(* IEC 61131-3 sources: SRCI/RobotLibrary/Library/Functions/Convert, 17 files *)

(* ---- ByteToFragmentAction.st ---- *)
FUNCTION ByteToFragmentAction : FragmentAction
// -------------------------------------------------------------------------
//  SRCI Robot Library
// -------------------------------------------------------------------------
//
//  Object:      FragmentActionToByte
//  Author:      Thorsten Brach
//  Date:        2024-11-05
//
//  Description:
//
//
//  Copyright:
//    (C) 2024 Thorsten Brach. All rights reserved
//             Licensed under the LGPL-3.0 license.
//
//  Disclaimer:
//    This project is provided without any guarantee and can be used for
//    private and commercial purposes. Any use is at the user’s
//    own risk and responsibility.
//
// -------------------------------------------------------------------------
VAR_INPUT
  FragmentAction : BYTE;
END_VAR

  ByteToFragmentAction.Complete:= FragmentAction.0;
  ByteToFragmentAction.Reset   := FragmentAction.1;
  ByteToFragmentAction.Clear   := FragmentAction.2;
  ByteToFragmentAction.BIT03   := FragmentAction.3;
  ByteToFragmentAction.BIT04   := FragmentAction.4;
  ByteToFragmentAction.BIT05   := FragmentAction.5;
  ByteToFragmentAction.BIT06   := FragmentAction.6;
  ByteToFragmentAction.BIT07   := FragmentAction.7;

END_FUNCTION

(* ---- CmdMessageStateToString.st ---- *)
FUNCTION CmdMessageStateToString : STRING
// -------------------------------------------------------------------------
//  SRCI Robot Library
// -------------------------------------------------------------------------
//
//  Object:      CmdMessageStateToString
//  Author:      Thorsten Brach
//  Date:        2024-11-16
//
//  Description:
//
//
//  Copyright:
//    (C) 2024 Thorsten Brach. All rights reserved
//             Licensed under the LGPL-3.0 license.
//
//  Disclaimer:
//    This project is provided without any guarantee and can be used for
//    private and commercial purposes. Any use is at the user’s
//    own risk and responsibility.
//
// -------------------------------------------------------------------------
VAR_INPUT
  /// Command message state
  Value : CmdMessageState;
END_VAR

  CASE Value
  OF
    CmdMessageState.EMPTY               : CmdMessageStateToString := StrReplace('EMPTY ({0})'              ,'{0}', USINT_TO_STRING(CmdMessageState.EMPTY));
    CmdMessageState.CREATED             : CmdMessageStateToString := StrReplace('CREATED ({0})'            ,'{0}', USINT_TO_STRING(CmdMessageState.CREATED));
    CmdMessageState.BUFFERED            : CmdMessageStateToString := StrReplace('BUFFERED ({0})'           ,'{0}', USINT_TO_STRING(CmdMessageState.BUFFERED));
    CmdMessageState.BUFFERED_IN_PLANNER : CmdMessageStateToString := StrReplace('BUFFERED_IN_PLANNER ({0})','{0}', USINT_TO_STRING(CmdMessageState.BUFFERED_IN_PLANNER));
    CmdMessageState.ACTIVE              : CmdMessageStateToString := StrReplace('ACTIVE ({0})'             ,'{0}', USINT_TO_STRING(CmdMessageState.ACTIVE));
    CmdMessageState.INTERRUPTED         : CmdMessageStateToString := StrReplace('INTERRUPTED ({0})'        ,'{0}', USINT_TO_STRING(CmdMessageState.INTERRUPTED));
    CmdMessageState.ABORT_REQUEST       : CmdMessageStateToString := StrReplace('ABORT_REQUEST ({0})'      ,'{0}', USINT_TO_STRING(CmdMessageState.ABORT_REQUEST));
    CmdMessageState.DONE                : CmdMessageStateToString := StrReplace('DONE ({0})'               ,'{0}', USINT_TO_STRING(CmdMessageState.DONE));
    CmdMessageState.ABORTED             : CmdMessageStateToString := StrReplace('ABORTED ({0})'            ,'{0}', USINT_TO_STRING(CmdMessageState.ABORTED));
    CmdMessageState.ERROR               : CmdMessageStateToString := StrReplace('ERROR ({0})'              ,'{0}', USINT_TO_STRING(CmdMessageState.ERROR));
  ELSE
    CmdMessageStateToString := CONCAT('CmdMessageStateToString-Function: Error -> no parsing for value ', USINT_TO_STRING(Value));
  END_CASE

END_FUNCTION

(* ---- CmdTypeToString.st ---- *)
FUNCTION CmdTypeToString : String
// -------------------------------------------------------------------------
//  SRCI Robot Library
// -------------------------------------------------------------------------
//
//  Object:      CmdTypeToString
//  Author:      Thorsten Brach
//  Date:        2024-11-16
//
//  Description:
//
//
//  Copyright:
//    (C) 2024 Thorsten Brach. All rights reserved
//             Licensed under the LGPL-3.0 license.
//
//  Disclaimer:
//    This project is provided without any guarantee and can be used for
//    private and commercial purposes. Any use is at the user’s
//    own risk and responsibility.
//
// -------------------------------------------------------------------------
VAR_INPUT
  /// command type
  Value : CmdType;
END_VAR

  CASE Value
  OF
    CmdType.RobotTask                   : CmdTypeToString := StrReplace('RobotTask ({0})','{0}'                  , UINT_TO_STRING(CmdType.RobotTask));

    CmdType.ReadRobotData               : CmdTypeToString := StrReplace('ReadRobotData ({0})','{0}'              , UINT_TO_STRING(CmdType.ReadRobotData));

    CmdType.EnableRobot                 : CmdTypeToString := StrReplace('EnableRobot ({0})','{0}'                , UINT_TO_STRING(CmdType.EnableRobot));

    CmdType.GroupReset                  : CmdTypeToString := StrReplace('GroupReset ({0})','{0}'                 , UINT_TO_STRING(CmdType.GroupReset));

    CmdType.ReadActualPosition          : CmdTypeToString := StrReplace('ReadActualPosition ({0})','{0}'         , UINT_TO_STRING(CmdType.ReadActualPosition));

    CmdType.ReadActualPositionCyclic    : CmdTypeToString := StrReplace('ReadActualPositionCyclic ({0})','{0}'   , UINT_TO_STRING(CmdType.ReadActualPositionCyclic));

    CmdType.ReadDHParameter             : CmdTypeToString := StrReplace('ReadDHParameter ({0})','{0}'            , UINT_TO_STRING(CmdType.ReadDHParameter));

    CmdType.RestartController           : CmdTypeToString := StrReplace('RestartController ({0})','{0}'          , UINT_TO_STRING(CmdType.RestartController));

    CmdType.ReadActualTCPVelocity       : CmdTypeToString := StrReplace('ReadActualTCPVelocity ({0})','{0}'      , UINT_TO_STRING(CmdType.ReadActualTCPVelocity));

    CmdType.UserLogin                   : CmdTypeToString := StrReplace('UserLogin ({0})','{0}'                  , UINT_TO_STRING(CmdType.UserLogin));

    CmdType.SwitchLanguage              : CmdTypeToString := StrReplace('SwitchLanguage ({0})','{0}'             , UINT_TO_STRING(CmdType.SwitchLanguage));

    CmdType.ExchangeConfiguration       : CmdTypeToString := StrReplace('ExchangeConfiguration ({0})','{0}'      , UINT_TO_STRING(CmdType.ExchangeConfiguration));

    CmdType.SetSequence                 : CmdTypeToString := StrReplace('SetSequence ({0})','{0}'                , UINT_TO_STRING(CmdType.SetSequence));

    CmdType.ChangeSpeedOverride         : CmdTypeToString := StrReplace('ChangeSpeedOverride ({0})','{0}'        , UINT_TO_STRING(CmdType.ChangeSpeedOverride));

    CmdType.ReadMessages                : CmdTypeToString := StrReplace('ReadMessages ({0})','{0}'               , UINT_TO_STRING(CmdType.ReadMessages));

    CmdType.ReadRobotReferenceDynamics  : CmdTypeToString := StrReplace('ReadRobotReferenceDynamics ({0})','{0}' , UINT_TO_STRING(CmdType.ReadRobotReferenceDynamics));

    CmdType.WriteFrameData              : CmdTypeToString := StrReplace('WriteFrameData ({0})','{0}'             , UINT_TO_STRING(CmdType.WriteFrameData));

    CmdType.WriteToolData               : CmdTypeToString := StrReplace('WriteToolData ({0})','{0}'              , UINT_TO_STRING(CmdType.WriteToolData));

    CmdType.WriteLoadData               : CmdTypeToString := StrReplace('WriteLoadData ({0})','{0}'              , UINT_TO_STRING(CmdType.WriteLoadData));

    CmdType.WriteRobotReferenceDynamics : CmdTypeToString := StrReplace('WriteRobotReferenceDynamics ({0})','{0}', UINT_TO_STRING(CmdType.WriteRobotReferenceDynamics));

    CmdType.WriteRobotDefaultDynamics   : CmdTypeToString := StrReplace('WriteRobotDefaultDynamics ({0})'  ,'{0}', UINT_TO_STRING(CmdType.WriteRobotDefaultDynamics));

    CmdType.ReadRobotDefaultDynamics    : CmdTypeToString := StrReplace('ReadRobotDefaultDynamics ({0})'   ,'{0}', UINT_TO_STRING(CmdType.ReadRobotDefaultDynamics));

    CmdType.ReadFrameData               : CmdTypeToString := StrReplace('ReadFrameData ({0})'              ,'{0}', UINT_TO_STRING(CmdType.ReadFrameData));

    CmdType.ReadToolData                : CmdTypeToString := StrReplace('ReadToolData ({0})','{0}'               , UINT_TO_STRING(CmdType.ReadToolData));

    CmdType.ReadLoadData                : CmdTypeToString := StrReplace('ReadLoadData ({0})','{0}'               , UINT_TO_STRING(CmdType.ReadLoadData));

    CmdType.ReadRobotSWLimits           : CmdTypeToString := StrReplace('ReadRobotSWLimits ({0})','{0}'          , UINT_TO_STRING(CmdType.ReadRobotSWLimits));

    CmdType.WriteRobotSWLimits          : CmdTypeToString := StrReplace('WriteRobotSWLimits ({0})','{0}'         , UINT_TO_STRING(CmdType.WriteRobotSWLimits));

    CmdType.SetOperationMode            : CmdTypeToString := StrReplace('SetOperationMode ({0})','{0}'           , UINT_TO_STRING(CmdType.SetOperationMode));

    CmdType.ReadWorkArea                : CmdTypeToString := StrReplace('ReadWorkArea ({0})','{0}'               , UINT_TO_STRING(CmdType.ReadWorkArea));

    CmdType.WriteWorkArea               : CmdTypeToString := StrReplace('WriteWorkArea ({0})','{0}'              , UINT_TO_STRING(CmdType.WriteWorkArea));

    CmdType.ActivateWorkArea            : CmdTypeToString := StrReplace('ActivateWorkArea ({0})','{0}'           , UINT_TO_STRING(CmdType.ActivateWorkArea));

    CmdType.MonitorWorkArea             : CmdTypeToString := StrReplace('MonitorWorkArea ({0})','{0}'            , UINT_TO_STRING(CmdType.MonitorWorkArea));

    CmdType.GroupJog                    : CmdTypeToString := StrReplace('GroupJog ({0})','{0}'                   , UINT_TO_STRING(CmdType.GroupJog));

    CmdType.MoveLinearAbsolute          : CmdTypeToString := StrReplace('MoveLinearAbsolute ({0})','{0}'         , UINT_TO_STRING(CmdType.MoveLinearAbsolute));

    CmdType.MoveDirectAbsolute          : CmdTypeToString := StrReplace('MoveDirectAbsolute ({0})','{0}'         , UINT_TO_STRING(CmdType.MoveDirectAbsolute));

    CmdType.MoveAxesAbsolute            : CmdTypeToString := StrReplace('MoveAxesAbsolute ({0})','{0}'           , UINT_TO_STRING(CmdType.MoveAxesAbsolute));

    CmdType.GroupStop                   : CmdTypeToString := StrReplace('GroupStop ({0})','{0}'                  , UINT_TO_STRING(CmdType.GroupStop));

    CmdType.GroupInterrupt              : CmdTypeToString := StrReplace('GroupInterrupt ({0})','{0}'             , UINT_TO_STRING(CmdType.GroupInterrupt));

    CmdType.GroupContinue               : CmdTypeToString := StrReplace('GroupContinue ({0})','{0}'              , UINT_TO_STRING(CmdType.GroupContinue));

    CmdType.MoveLinearRelative          : CmdTypeToString := StrReplace('MoveLinearRelative ({0})','{0}'         , UINT_TO_STRING(CmdType.MoveLinearRelative));

    CmdType.MoveDirectRelative          : CmdTypeToString := StrReplace('MoveDirectRelative ({0})','{0}'         , UINT_TO_STRING(CmdType.MoveDirectRelative));

    CmdType.MoveAxesRelative            : CmdTypeToString := StrReplace('MoveAxesRelative ({0})','{0}'           , UINT_TO_STRING(CmdType.MoveAxesRelative));

    CmdType.ReturnToPrimary             : CmdTypeToString := StrReplace('ReturnToPrimary ({0})','{0}'            , UINT_TO_STRING(CmdType.ReturnToPrimary));

    CmdType.MoveCircularAbsolute        : CmdTypeToString := StrReplace('MoveCircularAbsolute ({0})','{0}'       , UINT_TO_STRING(CmdType.MoveCircularAbsolute));

    CmdType.MoveCircularRelative        : CmdTypeToString := StrReplace('MoveCircularRelative ({0})','{0}'       , UINT_TO_STRING(CmdType.MoveCircularRelative));

    CmdType.MoveLinearOffset            : CmdTypeToString := StrReplace('MoveLinearOffset ({0})','{0}'           , UINT_TO_STRING(CmdType.MoveLinearOffset));

    CmdType.MoveDirectOffset            : CmdTypeToString := StrReplace('MoveDirectOffset ({0})','{0}'           , UINT_TO_STRING(CmdType.MoveDirectOffset));

    CmdType.WaitTime                    : CmdTypeToString := StrReplace('WaitTime ({0})','{0}'                   , UINT_TO_STRING(CmdType.WaitTime));

    CmdType.MoveApproachLinear          : CmdTypeToString := StrReplace('MoveApproachLinear ({0})','{0}'         , UINT_TO_STRING(CmdType.MoveApproachLinear));

    CmdType.MoveDepartLinear            : CmdTypeToString := StrReplace('MoveDepartLinear ({0})','{0}'           , UINT_TO_STRING(CmdType.MoveDepartLinear));

    CmdType.MoveApproachDirect          : CmdTypeToString := StrReplace('MoveApproachDirect ({0})','{0}'         , UINT_TO_STRING(CmdType.MoveApproachDirect));

    CmdType.MoveDepartDirect            : CmdTypeToString := StrReplace('MoveDepartDirect ({0})','{0}'           , UINT_TO_STRING(CmdType.MoveDepartDirect));

    CmdType.SearchHardstop              : CmdTypeToString := StrReplace('SearchHardstop ({0})','{0}'             , UINT_TO_STRING(CmdType.SearchHardstop));

    CmdType.SearchHardstopJ             : CmdTypeToString := StrReplace('SearchHardstopJ ({0})','{0}'            , UINT_TO_STRING(CmdType.SearchHardstopJ));

    CmdType.MovePickPlaceLinear         : CmdTypeToString := StrReplace('MovePickPlaceLinear ({0})','{0}'        , UINT_TO_STRING(CmdType.MovePickPlaceLinear));

    CmdType.MovePickPlaceDirect         : CmdTypeToString := StrReplace('MovePickPlaceDirect ({0})','{0}'        , UINT_TO_STRING(CmdType.MovePickPlaceDirect));

    CmdType.ActivateConveyorTracking    : CmdTypeToString := StrReplace('ActivateConveyorTracking ({0})','{0}'   , UINT_TO_STRING(CmdType.ActivateConveyorTracking));

    CmdType.RedefineTrackingPos         : CmdTypeToString := StrReplace('RedefineTrackingPos ({0})','{0}'        , UINT_TO_STRING(CmdType.RedefineTrackingPos));

    CmdType.SyncToConveyor              : CmdTypeToString := StrReplace('SyncToConveyor ({0})','{0}'             , UINT_TO_STRING(CmdType.SyncToConveyor));

    CmdType.ConfigureConveyor           : CmdTypeToString := StrReplace('ConfigureConveyor ({0})','{0}'          , UINT_TO_STRING(CmdType.ConfigureConveyor));

    CmdType.MoveSuperImposed            : CmdTypeToString := StrReplace('MoveSuperImposed ({0})','{0}'           , UINT_TO_STRING(CmdType.MoveSuperImposed));

    CmdType.MoveSuperImposedDynamic     : CmdTypeToString := StrReplace('MoveSuperImposedDynamic ({0})','{0}'    , UINT_TO_STRING(CmdType.MoveSuperImposedDynamic));

    CmdType.ReadDigitalInputs           : CmdTypeToString := StrReplace('ReadDigitalInputs ({0})','{0}'          , UINT_TO_STRING(CmdType.ReadDigitalInputs));

    CmdType.ReadDigitalOutputs          : CmdTypeToString := StrReplace('ReadDigitalOutputs ({0})','{0}'         , UINT_TO_STRING(CmdType.ReadDigitalOutputs));

    CmdType.WriteDigitalOutputs         : CmdTypeToString := StrReplace('WriteDigitalOutputs ({0})','{0}'        , UINT_TO_STRING(CmdType.WriteDigitalOutputs));

    CmdType.ReadIntegers                : CmdTypeToString := StrReplace('ReadIntegers ({0})','{0}'               , UINT_TO_STRING(CmdType.ReadIntegers));

    CmdType.ReadReals                   : CmdTypeToString := StrReplace('ReadReals ({0})','{0}'                  , UINT_TO_STRING(CmdType.ReadReals));

    CmdType.WriteIntegers               : CmdTypeToString := StrReplace('WriteIntegers ({0})','{0}'              , UINT_TO_STRING(CmdType.WriteIntegers));

    CmdType.WriteReals                  : CmdTypeToString := StrReplace('WriteReals ({0})','{0}'                 , UINT_TO_STRING(CmdType.WriteReals));

    CmdType.MoveLinearCam               : CmdTypeToString := StrReplace('MoveLinearCam ({0})','{0}'              , UINT_TO_STRING(CmdType.MoveLinearCam));

    CmdType.MoveDirectCam               : CmdTypeToString := StrReplace('MoveDirectCam ({0})','{0}'              , UINT_TO_STRING(CmdType.MoveDirectCam));

    CmdType.MoveCircularCam             : CmdTypeToString := StrReplace('MoveCircularCam ({0})','{0}'            , UINT_TO_STRING(CmdType.MoveCircularCam));

    CmdType.ReadAnalogInput             : CmdTypeToString := StrReplace('ReadAnalogInput ({0})','{0}'            , UINT_TO_STRING(CmdType.ReadAnalogInput));

    CmdType.ReadAnalogOutput            : CmdTypeToString := StrReplace('ReadAnalogOutput ({0})','{0}'           , UINT_TO_STRING(CmdType.ReadAnalogOutput));

    CmdType.WriteAnalogOutput           : CmdTypeToString := StrReplace('WriteAnalogOutput ({0})','{0}'          , UINT_TO_STRING(CmdType.WriteAnalogOutput));

    CmdType.MeasuringInput              : CmdTypeToString := StrReplace('MeasuringInput ({0})','{0}'             , UINT_TO_STRING(CmdType.MeasuringInput));

    CmdType.AbortMeasuringInput         : CmdTypeToString := StrReplace('AbortMeasuringInput ({0})','{0}'        , UINT_TO_STRING(CmdType.AbortMeasuringInput));

    CmdType.SetTriggerRegister          : CmdTypeToString := StrReplace('SetTriggerRegister ({0})','{0}'         , UINT_TO_STRING(CmdType.SetTriggerRegister));

    CmdType.SetTriggerLimit             : CmdTypeToString := StrReplace('SetTriggerLimit ({0})','{0}'            , UINT_TO_STRING(CmdType.SetTriggerLimit));

    CmdType.SetTriggerUser              : CmdTypeToString := StrReplace('SetTriggerUser ({0})','{0}'             , UINT_TO_STRING(CmdType.SetTriggerUser));

    CmdType.SetTriggerError             : CmdTypeToString := StrReplace('SetTriggerError ({0})','{0}'            , UINT_TO_STRING(CmdType.SetTriggerError));

    CmdType.ReactAtTrigger              : CmdTypeToString := StrReplace('ReactAtTrigger ({0})','{0}'             , UINT_TO_STRING(CmdType.ReactAtTrigger));

    CmdType.WaitForTrigger              : CmdTypeToString := StrReplace('WaitForTrigger ({0})','{0}'             , UINT_TO_STRING(CmdType.WaitForTrigger));

    CmdType.ReadSystemVariable          : CmdTypeToString := StrReplace('ReadSystemVariable ({0})','{0}'         , UINT_TO_STRING(CmdType.ReadSystemVariable));

    CmdType.WriteSystemVariable         : CmdTypeToString := StrReplace('WriteSystemVariable ({0})','{0}'        , UINT_TO_STRING(CmdType.WriteSystemVariable));

    CmdType.CalculateForwardKinematic   : CmdTypeToString := StrReplace('CalculateForwardKinematic ({0})','{0}'  , UINT_TO_STRING(CmdType.CalculateForwardKinematic));

    CmdType.CalculateInverseKinematic   : CmdTypeToString := StrReplace('CalculateInverseKinematic ({0})','{0}'  , UINT_TO_STRING(CmdType.CalculateInverseKinematic));

    CmdType.CalculateCartesianPosition  : CmdTypeToString := StrReplace('CalculateCartesianPosition ({0})','{0}' , UINT_TO_STRING(CmdType.CalculateCartesianPosition));

    CmdType.CalculateTool               : CmdTypeToString := StrReplace('CalculateTool ({0})','{0}'              , UINT_TO_STRING(CmdType.CalculateTool));

    CmdType.CalculateFrame              : CmdTypeToString := StrReplace('CalculateFrame ({0})','{0}'             , UINT_TO_STRING(CmdType.CalculateFrame));

    CmdType.ActivateNextCommand         : CmdTypeToString := StrReplace('ActivateNextCommand ({0})','{0}'        , UINT_TO_STRING(CmdType.ActivateNextCommand));

    CmdType.ShiftPosition               : CmdTypeToString := StrReplace('ShiftPosition ({0})','{0}'              , UINT_TO_STRING(CmdType.ShiftPosition));

    CmdType.SetTriggerMotion            : CmdTypeToString := StrReplace('SetTriggerMotion ({0})','{0}'           , UINT_TO_STRING(CmdType.SetTriggerMotion));

    CmdType.OpenBrake                   : CmdTypeToString := StrReplace('OpenBrake ({0})','{0}'                  , UINT_TO_STRING(CmdType.OpenBrake));

    CmdType.CallSubprogram              : CmdTypeToString := StrReplace('CallSubprogram ({0})','{0}'             , UINT_TO_STRING(CmdType.CallSubprogram));

    CmdType.WriteCallSubprogramCyclic   : CmdTypeToString := StrReplace('WriteCallSubprogramCyclic ({0})','{0}'  , UINT_TO_STRING(CmdType.WriteCallSubprogramCyclic));

    CmdType.ReadCallSubprogramCyclic    : CmdTypeToString := StrReplace('ReadCallSubprogramCyclic ({0})','{0}'   , UINT_TO_STRING(CmdType.ReadCallSubprogramCyclic));

    CmdType.StopSubprogram              : CmdTypeToString := StrReplace('StopSubprogram ({0})','{0}'             , UINT_TO_STRING(CmdType.StopSubprogram));

    CmdType.PathAccuracyMode            : CmdTypeToString := StrReplace('PathAccuracyMode ({0})','{0}'           , UINT_TO_STRING(CmdType.PathAccuracyMode));

    CmdType.AvoidSingularity            : CmdTypeToString := StrReplace('AvoidSingularity ({0})','{0}'           , UINT_TO_STRING(CmdType.AvoidSingularity));

    CmdType.ForceControl                : CmdTypeToString := StrReplace('ForceControl ({0})','{0}'               , UINT_TO_STRING(CmdType.ForceControl));

    CmdType.ForceLimit                  : CmdTypeToString := StrReplace('ForceLimit ({0})','{0}'                 , UINT_TO_STRING(CmdType.ForceLimit));

    CmdType.ReadActualForce             : CmdTypeToString := StrReplace('ReadActualForce ({0})','{0}'            , UINT_TO_STRING(CmdType.ReadActualForce));

    CmdType.BrakeTest                   : CmdTypeToString := StrReplace('BrakeTest ({0})','{0}'                  , UINT_TO_STRING(CmdType.BrakeTest));

    CmdType.SoftSwitchTCP               : CmdTypeToString := StrReplace('SoftSwitchTCP ({0})','{0}'              , UINT_TO_STRING(CmdType.SoftSwitchTCP));

    CmdType.CreateSpline                : CmdTypeToString := StrReplace('CreateSpline ({0})','{0}'               , UINT_TO_STRING(CmdType.CreateSpline));

    CmdType.DeleteSpline                : CmdTypeToString := StrReplace('DeleteSpline ({0})','{0}'               , UINT_TO_STRING(CmdType.DeleteSpline));

    CmdType.MoveSpline                  : CmdTypeToString := StrReplace('MoveSpline ({0})','{0}'                 , UINT_TO_STRING(CmdType.MoveSpline));

    CmdType.DynamicSpline               : CmdTypeToString := StrReplace('DynamicSpline ({0})','{0}'              , UINT_TO_STRING(CmdType.DynamicSpline));

    CmdType.LoadMeasurementAutomatic    : CmdTypeToString := StrReplace('LoadMeasurementAutomatic ({0})','{0}'   , UINT_TO_STRING(CmdType.LoadMeasurementAutomatic));

    CmdType.LoadMeasurementSequential   : CmdTypeToString := StrReplace('LoadMeasurementSequential ({0})','{0}'  , UINT_TO_STRING(CmdType.LoadMeasurementSequential));

    CmdType.CollisionDetection          : CmdTypeToString := StrReplace('CollisionDetection ({0})','{0}'         , UINT_TO_STRING(CmdType.CollisionDetection));

    CmdType.FreeDrive                   : CmdTypeToString := StrReplace('FreeDrive ({0})','{0}'                  , UINT_TO_STRING(CmdType.FreeDrive));

    CmdType.UnitMeasurement             : CmdTypeToString := StrReplace('UnitMeasurement ({0})','{0}'            , UINT_TO_STRING(CmdType.UnitMeasurement));

  ELSE
    CmdTypeToString := CONCAT('CmdTypeToString-Function: Error -> no parsing for value',UINT_TO_STRING(Value));
  END_CASE

END_FUNCTION

(* ---- CombineHalfBytes.st ---- *)
FUNCTION CombineHalfBytes : USINT
// -------------------------------------------------------------------------
//  SRCI Robot Library
// -------------------------------------------------------------------------
//
//  Object:      CombineHalfBytes
//  Author:      Thorsten Brach
//  Date:        2024-06-01
//
//  Description:
//
//
//  Copyright:
//    (C) 2024 Thorsten Brach. All rights reserved
//             Licensed under the LGPL-3.0 license.
//
//  Disclaimer:
//    This project is provided without any guarantee and can be used for
//    private and commercial purposes. Any use is at the user’s
//    own risk and responsibility.
//
// -------------------------------------------------------------------------
VAR_INPUT
  /// Half-Byte to add to the upper 4 Bit
  HalfByteHi : BYTE;
  /// Half-Byte to add to the lower 4 Bit
  HalfByteLo : BYTE;
END_VAR

  // merage ParSeq and Priority to combined variable
  CombineHalfBytes.0 := HalfByteLo.0;
  CombineHalfBytes.1 := HalfByteLo.1;
  CombineHalfBytes.2 := HalfByteLo.2;
  CombineHalfBytes.3 := HalfByteLo.3;

  CombineHalfBytes.4 := HalfByteHi.0;
  CombineHalfBytes.5 := HalfByteHi.1;
  CombineHalfBytes.6 := HalfByteHi.2;
  CombineHalfBytes.7 := HalfByteHi.3;

END_FUNCTION

(* ---- DATE_TO_IEC_DATE.st ---- *)
FUNCTION DATE_TO_IEC_DATE : IEC_DATE
// -------------------------------------------------------------------------
//  SRCI Robot Library
// -------------------------------------------------------------------------
//
//  Object:      DATE_TO_IEC_DATE
//  Author:      Thorsten Brach
//  Date:        2024-06-01
//
//  Description:
//
//
//  Copyright:
//    (C) 2024 Thorsten Brach. All rights reserved
//             Licensed under the LGPL-3.0 license.
//
//  Disclaimer:
//    This project is provided without any guarantee and can be used for
//    private and commercial purposes. Any use is at the user’s
//    own risk and responsibility.
//
// -------------------------------------------------------------------------
VAR_INPUT
  Value    : DATE;
END_VAR

VAR
 _tmpDate1 : DWORD;
 _tmpDate2 : DWORD;
 _initDate : DATE := DATE#1990-01-01;
 END_VAR

  /// Siemens Dateformat is Day since 01.01.1990
  /// TwinCat Dateformat is seconds sinde 01.01.1970
  /// Calculation :
  /// ( [TwinCat current date] - [ TwinCat 01.01.1970] ) / [Seconds a Day] = Days sinde 01.01.1990 (Siemens Format)

  /// copy date to dword
  SysDepMemCpy( pDest := ADR(_tmpDate1), pSrc := ADR( Value   ), DataLen := SIZEOF( Value   ));
  /// copy date to dword
  SysDepMemCpy( pDest := ADR(_tmpDate2), pSrc := ADR(_initDate), DataLen := SIZEOF(_initDate));

  /// calculate IEC Date :
  DATE_TO_IEC_DATE := UDINT_TO_UINT((_tmpDate1 - _tmpDate2) / 86400); // 86400 Seconds = 1 day

END_FUNCTION

(* ---- FragmentActionToByte.st ---- *)
FUNCTION FragmentActionToByte : BYTE
// -------------------------------------------------------------------------
//  SRCI Robot Library
// -------------------------------------------------------------------------
//
//  Object:      FragmentActionToByte
//  Author:      Thorsten Brach
//  Date:        2024-06-01
//
//  Description:
//
//
//  Copyright:
//    (C) 2024 Thorsten Brach. All rights reserved
//             Licensed under the LGPL-3.0 license.
//
//  Disclaimer:
//    This project is provided without any guarantee and can be used for
//    private and commercial purposes. Any use is at the user’s
//    own risk and responsibility.
//
// -------------------------------------------------------------------------
VAR_INPUT
  FragmentAction : FragmentAction;
END_VAR

  FragmentActionToByte.0 := FragmentAction.Complete;
  FragmentActionToByte.1 := FragmentAction.Reset;
  FragmentActionToByte.2 := FragmentAction.Clear;
  FragmentActionToByte.3 := FragmentAction.BIT03;
  FragmentActionToByte.4 := FragmentAction.BIT04;
  FragmentActionToByte.5 := FragmentAction.BIT05;
  FragmentActionToByte.6 := FragmentAction.BIT06;
  FragmentActionToByte.7 := FragmentAction.BIT07;

END_FUNCTION

(* ---- IEC_DATE_TO_DATE.st ---- *)
FUNCTION IEC_DATE_TO_DATE : DATE
// -------------------------------------------------------------------------
//  SRCI Robot Library
// -------------------------------------------------------------------------
//
//  Object:      IEC_DATE_TO_DATE
//  Author:      Thorsten Brach
//  Date:        2025-01-05
//
//  Description:
//
//
//  Copyright:
//    (C) 2025 Thorsten Brach. All rights reserved
//             Licensed under the LGPL-3.0 license.
//
//  Disclaimer:
//    This project is provided without any guarantee and can be used for
//    private and commercial purposes. Any use is at the user’s
//    own risk and responsibility.
//
// -------------------------------------------------------------------------
VAR_INPUT
  Value    : IEC_DATE;
END_VAR

VAR
 _tmpDate1 : DWORD;
 _initDate : DATE := DATE#1990-01-01;
 END_VAR

  // Siemens Dateformat is Day since 01.01.1990
  // TwinCat Dateformat is seconds sinde 01.01.1970
  // Calculation :
  // ( [ TwinCat 01.01.1990] + [IEC Date]) * [Seconds a Day] = (TwinCat Format)

  // copy date to dword
  SysDepMemCpy( pDest := ADR(_tmpDate1), pSrc := ADR( _initDate ), DataLen := SIZEOF( _initDate ));

  // calculate IEC Date :
  IEC_DATE_TO_DATE := DWORD_TO_DATE( _tmpDate1 + ( Value * 86400)); // 86400 Seconds = 1 day

END_FUNCTION

(* ---- IEC_TIME_TO_TIME.st ---- *)
FUNCTION IEC_TIME_TO_TIME : TOD
// -------------------------------------------------------------------------
//  SRCI Robot Library
// -------------------------------------------------------------------------
//
//  Object:      IEC_TIME_TO_TIME
//  Author:      Thorsten Brach
//  Date:        2025-01-05
//
//  Description:
//
//
//  Copyright:
//    (C) 2025 Thorsten Brach. All rights reserved
//             Licensed under the LGPL-3.0 license.
//
//  Disclaimer:
//    This project is provided without any guarantee and can be used for
//    private and commercial purposes. Any use is at the user’s
//    own risk and responsibility.
//
// -------------------------------------------------------------------------
VAR_INPUT
  Value : IEC_TIME;
END_VAR

  IEC_TIME_TO_TIME := Value;

END_FUNCTION

(* ---- MESSAGE_TYPE_TO_STRING.st ---- *)
FUNCTION MESSAGE_TYPE_TO_STRING : STRING
// -------------------------------------------------------------------------
//  SRCI Robot Library
// -------------------------------------------------------------------------
//
//  Object:      MESSAGE_TYPE_TO_STRING
//  Author:      Thorsten Brach
//  Date:        2025-01-11
//
//  Description:
//
//
//  Copyright:
//    (C) 2025 Thorsten Brach. All rights reserved
//             Licensed under the LGPL-3.0 license.
//
//  Disclaimer:
//    This project is provided without any guarantee and can be used for
//    private and commercial purposes. Any use is at the user’s
//    own risk and responsibility.
//
// -------------------------------------------------------------------------
VAR_INPUT
  /// Severity
  Value     : MessageType;
  /// Fill spaces to the end, so that all values has the same length
  AlignString : BOOL;
END_VAR

  IF (AlignString)
  THEN
    CASE Value OF

      MessageType.RI  : MESSAGE_TYPE_TO_STRING := 'RI ';
      MessageType.RC  : MESSAGE_TYPE_TO_STRING := 'RC ';
      MessageType.RA  : MESSAGE_TYPE_TO_STRING := 'RA ';
      MessageType.CMD : MESSAGE_TYPE_TO_STRING := 'CMD' ;
    ELSE
      MESSAGE_TYPE_TO_STRING := '???';
    END_CASE
  ELSE
    CASE Value OF

      MessageType.RI  : MESSAGE_TYPE_TO_STRING := 'RI';
      MessageType.RC  : MESSAGE_TYPE_TO_STRING := 'RC';
      MessageType.RA  : MESSAGE_TYPE_TO_STRING := 'RA';
      MessageType.CMD : MESSAGE_TYPE_TO_STRING := 'CMD' ;
    ELSE
      MESSAGE_TYPE_TO_STRING := '???';
    END_CASE
  END_IF

END_FUNCTION

(* ---- PlcOptionalCyclicToUint.st ---- *)
FUNCTION PlcOptionalCyclicToUint : UINT
// -------------------------------------------------------------------------
//  SRCI Robot Library
// -------------------------------------------------------------------------
//
//  Object:      PlcOptionalCyclicToUint
//  Author:      Thorsten Brach
//  Date:        2024-11-30
//
//  Description:
//
//
//  Copyright:
//    (C) 2024 Thorsten Brach. All rights reserved
//             Licensed under the LGPL-3.0 license.
//
//  Disclaimer:
//    This project is provided without any guarantee and can be used for
//    private and commercial purposes. Any use is at the user’s
//    own risk and responsibility.
//
// -------------------------------------------------------------------------
VAR_INPUT
  OptionalCyclic : AxesGroupParameterPlcOptionalCyclic;
END_VAR

  PlcOptionalCyclicToUint.00 := OptionalCyclic.UseCallSubprogram;
  PlcOptionalCyclicToUint.01 := OptionalCyclic.UseCartesianPosition;
  PlcOptionalCyclicToUint.02 := OptionalCyclic.UseJointPosition;
  PlcOptionalCyclicToUint.03 := OptionalCyclic.UseForce;
  PlcOptionalCyclicToUint.04 := OptionalCyclic.Bit04;
  PlcOptionalCyclicToUint.05 := OptionalCyclic.Bit05;
  PlcOptionalCyclicToUint.06 := OptionalCyclic.Bit06;
  PlcOptionalCyclicToUint.07 := OptionalCyclic.Bit07;
  PlcOptionalCyclicToUint.08 := OptionalCyclic.UseTwoSequences;
  PlcOptionalCyclicToUint.09 := OptionalCyclic.UseCartesianPositionExt;
  PlcOptionalCyclicToUint.10 := OptionalCyclic.UseJointPositionExt;
  PlcOptionalCyclicToUint.11 := OptionalCyclic.Bit11;
  PlcOptionalCyclicToUint.12 := OptionalCyclic.Bit12;
  PlcOptionalCyclicToUint.13 := OptionalCyclic.Bit13;
  PlcOptionalCyclicToUint.14 := OptionalCyclic.Bit14;
  PlcOptionalCyclicToUint.15 := OptionalCyclic.Bit15;

END_FUNCTION

(* ---- RobOptionalCyclicToUint.st ---- *)
FUNCTION RobOptionalCyclicToUint : UINT
// -------------------------------------------------------------------------
//  SRCI Robot Library
// -------------------------------------------------------------------------
//
//  Object:      RobOptionalCyclicToUint
//  Author:      Thorsten Brach
//  Date:        2024-11-30
//
//  Description:
//
//
//  Copyright:
//    (C) 2024 Thorsten Brach. All rights reserved
//             Licensed under the LGPL-3.0 license.
//
//  Disclaimer:
//    This project is provided without any guarantee and can be used for
//    private and commercial purposes. Any use is at the user’s
//    own risk and responsibility.
//
// -------------------------------------------------------------------------
VAR_INPUT
  OptionalCyclic : AxesGroupParameterRobOptionalCyclic;
END_VAR

  RobOptionalCyclicToUint.00 := OptionalCyclic.UseCallSubprogram;
  RobOptionalCyclicToUint.01 := OptionalCyclic.UseCartesianPosition;
  RobOptionalCyclicToUint.02 := OptionalCyclic.UseJointPosition;
  RobOptionalCyclicToUint.03 := OptionalCyclic.UseForce;
  RobOptionalCyclicToUint.04 := OptionalCyclic.UseCurrent;
  RobOptionalCyclicToUint.05 := OptionalCyclic.Bit05;
  RobOptionalCyclicToUint.06 := OptionalCyclic.Bit06;
  RobOptionalCyclicToUint.07 := OptionalCyclic.Bit07;
  RobOptionalCyclicToUint.08 := OptionalCyclic.UseTwoSequences;
  RobOptionalCyclicToUint.09 := OptionalCyclic.UseCartesianPositionExt;
  RobOptionalCyclicToUint.10 := OptionalCyclic.UseJointPositionExt;
  RobOptionalCyclicToUint.11 := OptionalCyclic.UseForceExt;
  RobOptionalCyclicToUint.12 := OptionalCyclic.UseCurrentExt;
  RobOptionalCyclicToUint.13 := OptionalCyclic.Bit13;
  RobOptionalCyclicToUint.14 := OptionalCyclic.Bit14;
  RobOptionalCyclicToUint.15 := OptionalCyclic.Bit15;

END_FUNCTION

(* ---- SEVERITY_TO_STRING.st ---- *)
FUNCTION SEVERITY_TO_STRING : STRING
// -------------------------------------------------------------------------
//  SRCI Robot Library
// -------------------------------------------------------------------------
//
//  Object:      SEVERITY_TO_STRING
//  Author:      Thorsten Brach
//  Date:        2025-01-11
//
//  Description:
//
//
//  Copyright:
//    (C) 2025 Thorsten Brach. All rights reserved
//             Licensed under the LGPL-3.0 license.
//
//  Disclaimer:
//    This project is provided without any guarantee and can be used for
//    private and commercial purposes. Any use is at the user’s
//    own risk and responsibility.
//
// -------------------------------------------------------------------------
VAR_INPUT
  /// Severity
  Value : Severity;
  /// Fill spaces to the end, so that all values has the same length
  AlignString : BOOL;
END_VAR

  IF (AlignString)
  THEN
    CASE Value OF
      Severity.DEBUG       : SEVERITY_TO_STRING := 'DEBUG      ';
      Severity.INFO        : SEVERITY_TO_STRING := 'INFO       ';
      Severity.WARNING     : SEVERITY_TO_STRING := 'WARNING    ';
      Severity.ERROR       : SEVERITY_TO_STRING := 'ERROR      ' ;
      Severity.FATAL_ERROR : SEVERITY_TO_STRING := 'FATAL_ERROR' ;
    ELSE
      SEVERITY_TO_STRING := 'UNKOWN     ';
    END_CASE
  ELSE
    CASE Value OF
      Severity.DEBUG       : SEVERITY_TO_STRING := 'DEBUG';
      Severity.INFO        : SEVERITY_TO_STRING := 'INFO';
      Severity.WARNING     : SEVERITY_TO_STRING := 'WARNING';
      Severity.ERROR       : SEVERITY_TO_STRING := 'ERROR' ;
      Severity.FATAL_ERROR : SEVERITY_TO_STRING := 'FATAL_ERROR' ;
    ELSE
      SEVERITY_TO_STRING := 'UNKOWN';
    END_CASE
  END_IF

END_FUNCTION

(* ---- TelegramControlToString.st ---- *)
FUNCTION TelegramControlToString : STRING
// -------------------------------------------------------------------------
//  SRCI Robot Library
// -------------------------------------------------------------------------
//
//  Object:      TelegramControlToString
//  Author:      Thorsten Brach
//  Date:        2024-11-16
//
//  Description:
//
//
//  Copyright:
//    (C) 2024 Thorsten Brach. All rights reserved
//             Licensed under the LGPL-3.0 license.
//
//  Disclaimer:
//    This project is provided without any guarantee and can be used for
//    private and commercial purposes. Any use is at the user’s
//    own risk and responsibility.
//
// -------------------------------------------------------------------------
VAR_INPUT
  /// Telegram state
  Control : ControlHalfByte;
END_VAR

  CASE Control OF
    ControlHalfByte.NONE         : TelegramControlToString := StrReplace('NONE ({0})'        ,'{0}', USINT_TO_STRING(ControlHalfByte.NONE));
    ControlHalfByte.INITIALIZE   : TelegramControlToString := StrReplace('INITIALIZE ({0})'  ,'{0}', USINT_TO_STRING(ControlHalfByte.INITIALIZE));
    ControlHalfByte.RESUME       : TelegramControlToString := StrReplace('RESUME ({0})'      ,'{0}', USINT_TO_STRING(ControlHalfByte.RESUME));
    ControlHalfByte.RESET        : TelegramControlToString := StrReplace('RESET ({0})'       ,'{0}', USINT_TO_STRING(ControlHalfByte.RESET));
    ControlHalfByte.ACK_ERROR    : TelegramControlToString := StrReplace('ACK_ERROR ({0})'   ,'{0}', USINT_TO_STRING(ControlHalfByte.ACK_ERROR));
    ControlHalfByte.CLIENT_ERROR : TelegramControlToString := StrReplace('CLIENT_ERROR ({0})','{0}', USINT_TO_STRING(ControlHalfByte.CLIENT_ERROR));
  ELSE
    TelegramControlToString := CONCAT('TelegramControlToString-Function: Error -> no parsing for value ', BYTE_TO_STRING(Control));
  END_CASE

END_FUNCTION

(* ---- TelegramStateToString.st ---- *)
FUNCTION TelegramStateToString : STRING
// -------------------------------------------------------------------------
//  SRCI Robot Library
// -------------------------------------------------------------------------
//
//  Object:      TelegramStateToString
//  Author:      Thorsten Brach
//  Date:        2024-11-16
//
//  Description:
//
//
//  Copyright:
//    (C) 2024 Thorsten Brach. All rights reserved
//             Licensed under the LGPL-3.0 license.
//
//  Disclaimer:
//    This project is provided without any guarantee and can be used for
//    private and commercial purposes. Any use is at the user’s
//    own risk and responsibility.
//
// -------------------------------------------------------------------------
VAR_INPUT
  /// Telegram state
  State : TelegramState;
END_VAR

  CASE State OF

    TelegramState.UNDEFINED                : TelegramStateToString := StrReplace('UNDEFINED ({0})'               ,'{0}', USINT_TO_STRING(TelegramState.UNDEFINED));
    TelegramState.ERROR_161                : TelegramStateToString := StrReplace('ERROR_161 ({0})'               ,'{0}', USINT_TO_STRING(TelegramState.ERROR_161));
    TelegramState.ERROR_162                : TelegramStateToString := StrReplace('ERROR_162 ({0})'               ,'{0}', USINT_TO_STRING(TelegramState.ERROR_162));
    TelegramState.ERROR_163                : TelegramStateToString := StrReplace('ERROR_163 ({0})'               ,'{0}', USINT_TO_STRING(TelegramState.ERROR_163));
    TelegramState.ERROR_164                : TelegramStateToString := StrReplace('ERROR_164 ({0})'               ,'{0}', USINT_TO_STRING(TelegramState.ERROR_164));
    TelegramState.ERROR_165                : TelegramStateToString := StrReplace('ERROR_165 ({0})'               ,'{0}', USINT_TO_STRING(TelegramState.ERROR_165));
    TelegramState.ERROR_166                : TelegramStateToString := StrReplace('ERROR_166 ({0})'               ,'{0}', USINT_TO_STRING(TelegramState.ERROR_166));
    TelegramState.ERROR_167                : TelegramStateToString := StrReplace('ERROR_167 ({0})'               ,'{0}', USINT_TO_STRING(TelegramState.ERROR_167));
    TelegramState.ERROR_168                : TelegramStateToString := StrReplace('ERROR_168 ({0})'               ,'{0}', USINT_TO_STRING(TelegramState.ERROR_168));
    TelegramState.ERROR_169                : TelegramStateToString := StrReplace('ERROR_169 ({0})'               ,'{0}', USINT_TO_STRING(TelegramState.ERROR_169));
    TelegramState.ERROR_170                : TelegramStateToString := StrReplace('ERROR_170 ({0})'               ,'{0}', USINT_TO_STRING(TelegramState.ERROR_170));
    TelegramState.ERROR_171                : TelegramStateToString := StrReplace('ERROR_171 ({0})'               ,'{0}', USINT_TO_STRING(TelegramState.ERROR_171));
    TelegramState.ERROR_172                : TelegramStateToString := StrReplace('ERROR_172 ({0})'               ,'{0}', USINT_TO_STRING(TelegramState.ERROR_172));
    TelegramState.READY_TO_RESUME          : TelegramStateToString := StrReplace('READY_TO_RESUME ({0})'         ,'{0}', USINT_TO_STRING(TelegramState.READY_TO_RESUME));
    TelegramState.READY_FOR_INITIALIZATION : TelegramStateToString := StrReplace('READY_FOR_INITIALIZATION ({0})','{0}', USINT_TO_STRING(TelegramState.READY_FOR_INITIALIZATION));
    TelegramState.INITIALIZED              : TelegramStateToString := StrReplace('INITIALIZED ({0})'             ,'{0}', USINT_TO_STRING(TelegramState.INITIALIZED));
  ELSE
    TelegramStateToString := CONCAT('TelegramStateToString-Function: Error -> no parsing for value ', USINT_TO_STRING(State));
  END_CASE

END_FUNCTION

(* ---- WORD_TO_STRING_HEX.st ---- *)
FUNCTION WORD_TO_STRING_HEX : STRING
// -------------------------------------------------------------------------
//  SRCI Robot Library
// -------------------------------------------------------------------------
//
//  Object:      WORD_TO_STRING_HEX
//  Author:      Thorsten Brach
//  Date:        2024-12-13
//
//  Description:
//    Converts a WORD to a STRING with hex notation
//
//  Copyright:
//    (C) 2024 Thorsten Brach. All rights reserved
//             Licensed under the LGPL-3.0 license.
//
//  Disclaimer:
//    This project is provided without any guarantee and can be used for
//    private and commercial purposes. Any use is at the user’s
//    own risk and responsibility.
//
// -------------------------------------------------------------------------
VAR_INPUT
 /// Value to convert
 Value : WORD;
END_VAR
VAR
  /// high Byte
 _highByte   : BYTE;
  /// low Byte
 _lowByte    : BYTE;
  /// high Nibble
 _highNibble : BYTE;
  /// low Nibble
 _lowNibble  : BYTE;
  /// single Hex char
  hexChar    : STRING(1);
  /// Hex chars
  hexChars   : ARRAY[0..15] OF STRING(1) := ['0', '1', '2', '3', '4', '5', '6', '7', '8', '9', 'A', 'B', 'C', 'D', 'E', 'F'];
END_VAR

  // get high and low byte from word
  _highByte := WORD_TO_BYTE(SHR(Value, 8));
  _lowByte  := WORD_TO_BYTE(Value AND 16#FF);

  // convert highest Byte to HEX
  _highNibble := SHR(_highByte, 4);
  _lowNibble  := (_highByte AND 16#F);
  WORD_TO_STRING_HEX := CONCAT(hexChars[_highNibble], hexChars[_lowNibble]);

  // convert lowest Byte to HEX
  _highNibble := SHR(_lowByte, 4);
  _lowNibble := _lowByte AND 16#F;
  WORD_TO_STRING_HEX := CONCAT(WORD_TO_STRING_HEX, CONCAT(hexChars[_highNibble], hexChars[_lowNibble]));

END_FUNCTION

(* ---- WordToArmConfigElbow.st ---- *)
FUNCTION WordToArmConfigElbow : ArmConfigElbow
// -------------------------------------------------------------------------
//  SRCI Robot Library
// -------------------------------------------------------------------------
//
//  Object:      WordToArmConfigElbow
//  Author:      Thorsten Brach
//  Date:        2024-12-24
//
//  Description:
//
//
//  Copyright:
//    (C) 2024 Thorsten Brach. All rights reserved
//             Licensed under the LGPL-3.0 license.
//
//  Disclaimer:
//    This project is provided without any guarantee and can be used for
//    private and commercial purposes. Any use is at the user’s
//    own risk and responsibility.
//
// -------------------------------------------------------------------------
VAR_INPUT
  /// Value
  Value : WORD;
END_VAR

VAR
  _tmpByte : BYTE;
END_VAR

  IF (Value.1)
  THEN
    WordToArmConfigElbow := ArmConfigElbow.DOWN;
  ELSE
    WordToArmConfigElbow := ArmConfigElbow.UP;
  END_IF

END_FUNCTION

(* ---- WordToArmConfigWrist.st ---- *)
FUNCTION WordToArmConfigWrist : ArmConfigWrist
// -------------------------------------------------------------------------
//  SRCI Robot Library
// -------------------------------------------------------------------------
//
//  Object:      WordToArmConfigWrist
//  Author:      Thorsten Brach
//  Date:        2024-12-24
//
//  Description:
//
//
//  Copyright:
//    (C) 2024 Thorsten Brach. All rights reserved
//             Licensed under the LGPL-3.0 license.
//
//  Disclaimer:
//    This project is provided without any guarantee and can be used for
//    private and commercial purposes. Any use is at the user’s
//    own risk and responsibility.
//
// -------------------------------------------------------------------------
VAR_INPUT
  /// Value
  Value : WORD;
END_VAR

VAR
  _tmpByte : BYTE;
END_VAR

  IF (Value.2)
  THEN
    WordToArmConfigWrist := ArmConfigWrist.FLIP;
  ELSE
    WordToArmConfigWrist := ArmConfigWrist.NON_FLIP;
  END_IF

END_FUNCTION
